(*
Nazwa:			FB_ReadWriteCSV
Opis:			Zapis uzytkownikow do pliku CSV
Wersja:			v0.1
Data:			2018-10-31
Autor:			
Urzadzenia:		
Konfiguracja:	
Info:
*)
FUNCTION_BLOCK FB_ReadWriteLogCSV
VAR
	sCSVLine				: T_MaxString := '';(* Single CSV text line (row, record), we are using string as record buffer (your are able to see read fields)  *)
	sCSVField				: T_MaxString := '';(* Single CSV field value (column, record field) *)
	nRow	 				: UDINT 	:= 0;(* Row number (record) *)
	nColumn					: UDINT 	:= 0;(* Column number (record field) *)
	hFile					: UINT		:= 0;(* File handle of the source file *)
	step					: DWORD 	:= 0;
	fbFileOpen				: FB_FileOpen;(* Opens file *)
	fbFileClose				: FB_FileClose;(* Closes file *)
	fbFileGets				: FB_FileGets;(* Reads one record (line) *)
	fbReader				: FB_CSVMemBufferReader;(* Helper function block used to parse CSV data bytes (single record line) *)
	fbFilePuts				: FB_FilePuts;(* Writes one record (line) *)
	fbWriter				: FB_CSVMemBufferWriter;(* Helper function block used to create CSV data bytes (single record line) *)
	database				: ARRAY[0..239, 0..10] OF STRING(100);(* Target PLC database *)
	i						: INT;
	iNum					: INT;
	BusyFTRIG				: F_TRIG;	// Zakonczenie zapisu/odczytu pliku
	CommandRTRIG			: R_TRIG;	// Wykrycie zapisu/odczytu
	ErrorFileDataUsers		: R_TRIG;	// Błąd zapisu/odczytu
	bNewFile				: BOOL;		// Utworzenie nowego pliku
	iMode					: INT;		// Zapis/odczyt
	
	MAX_CSV_ROWS 			: UDINT := 239;
	MAX_CSV_COLUMNS 		: UDINT := 10;
	MAX_CSV_FIELD_LENGTH	: UDINT := 100;
	
//	fbGetDateTime			: NT_GetTime;
	sDateTime				: STRING[200];
	fbFileTell				: FB_FileTell;
	fbEOF					: FB_EOF;
	fbFileSeek				: FB_FileSeek;
	
	sLineToWrite			:STRING(255);
END_VAR
	
VAR_INPUT
	bRead					: BOOL;		//Sygnal odczytu pliku
	bWrite					: BOOL;		//Sygnal zapisu pliku
	stDataArray				: ARRAY [0..239] OF S_LogData;	//Tablica z danymi
	sNetId					: T_AmsNetId := '';	(* TwinCAT system network address *)
	sFileName				: T_MaxString ;(* CSV destination file path and name *)
END_VAR
VAR_OUTPUT
	bError					: BOOL;		// Sygnal błedu
	bBusy					: BOOL;		// Sygnal zajetosci
	bDone					: BOOL;		// Sygnal zakonczenia odczytu/zapisu
	nErrId					: UDINT;	// Numer bledu
END_VAR

CASE step OF
	0:	(* Wait for rising edge at bWrite variable *)
		IF bWrite (*AND NOT fbGetDateTime.BUSY*) THEN
			bWrite 		:= FALSE;
			bBusy 		:= TRUE;
			bError		:= FALSE;
			nErrId		:= 0;
			hFile		:= 0;
			nRow	 	:= 1;			//było 0
			nColumn		:= 0;
			step 		:= 1;
			//wybiera elementy do zapisania
			FOR iNum := 0 TO TO_INT(MAX_CSV_ROWS) DO
//				sDateTime			:=SYSTEMTIME_TO_STRING(fbGetDateTime.TIMESTR);
//				sDateTime			:=DELETE(sDateTime,11,1);	//Usuwa datę
//				sDateTime			:=LEFT(sDateTime,find(sDateTime,'.')-1); //usuwa licznik ms
				    


				//	sLineToWrite := CONCAT(WSTRING_TO_STRING(P_time.s_time_mainscreen), ',');
   		 		//	sLineToWrite := CONCAT(sLineToWrite, REAL_TO_STRING(P_ADS_SCREW.lrGripperScrewer1TorqueCV));
   		 		//	sLineToWrite := CONCAT(sLineToWrite, ',');
   		 		//	sLineToWrite := CONCAT(sLineToWrite, WSTRING_TO_STRING(gvl_recipe.s_recipe_name));
   		 		//	sLineToWrite := CONCAT(sLineToWrite, '$N');	




				database[iNum,0]		:= WSTRING_TO_STRING(P_time.s_time_mainscreen);
				database[iNum,1]		:= REAL_TO_STRING(stDataArray[iNum].arData[0]);
				database[iNum,2]		:= REAL_TO_STRING(stDataArray[iNum].arData[1]);
				database[iNum,3]		:= REAL_TO_STRING(stDataArray[iNum].arData[2]);
				database[iNum,4]		:= REAL_TO_STRING(stDataArray[iNum].arData[3]);
				database[iNum,5]		:= REAL_TO_STRING(stDataArray[iNum].arData[4]);
				database[iNum,6]		:= REAL_TO_STRING(stDataArray[iNum].arData[5]);
				database[iNum,7]		:= REAL_TO_STRING(stDataArray[iNum].arData[6]);
				database[iNum,8]		:= REAL_TO_STRING(stDataArray[iNum].arData[7]);
				database[iNum,9]		:= REAL_TO_STRING(stDataArray[iNum].arData[8]);
				database[iNum,10]		:= REAL_TO_STRING(stDataArray[iNum].arData[9]);
				
//				database[iNum,0]		:= GVL.arLogDataSave1[iNum].tTime;
//				database[iNum,1]		:= REAL_TO_STRING(GVL.arLogDataSave1[iNum].arData[0]);
//				database[iNum,2]		:= REAL_TO_STRING(GVL.arLogDataSave1[iNum].arData[1]);
//				database[iNum,3]		:= REAL_TO_STRING(GVL.arLogDataSave1[iNum].arData[2]);
//				database[iNum,4]		:= REAL_TO_STRING(GVL.arLogDataSave1[iNum].arData[3]);
//				database[iNum,5]		:= REAL_TO_STRING(GVL.arLogDataSave1[iNum].arData[4]);
//				database[iNum,6]		:= REAL_TO_STRING(GVL.arLogDataSave1[iNum].arData[5]);
//				database[iNum,7]		:= REAL_TO_STRING(GVL.arLogDataSave1[iNum].arData[6]);
//				database[iNum,8]		:= REAL_TO_STRING(GVL.arLogDataSave1[iNum].arData[7]);
//				database[iNum,9]		:= REAL_TO_STRING(GVL.arLogDataSave1[iNum].arData[8]);
//				database[iNum,10]		:= REAL_TO_STRING(GVL.arLogDataSave1[iNum].arData[9]);
			END_FOR
			//zmienia . na , żeby szybciej przetwarzać dane w excelu
//			FOR i:=1 TO UDINT_TO_INT(MAX_CSV_COLUMNS) BY 1 DO
//				database[1,i]:=REPLACE(database[1,i],',',1,FIND(database[1,i],'.'));
//			END_FOR
		END_IF
	1:	(* Open source file *)
		fbFileOpen(bExecute := FALSE);
		fbFiletell(bExecute := FALSE);	//potrzebne do wykrycia nowego pliku
	//	fbEOF(bExecute:=FALSE);
		fbFileSeek(bExecute:=FALSE);	//potrzebne do wykrycia nowego pliku
		fbFileOpen( 	sNetId := sNetId, sPathName := sFileName, nMode := FOPEN_MODEAPPEND OR FOPEN_MODETEXT,(* Open file in TEXT mode! *)
						ePath := PATH_GENERIC, bExecute := TRUE );
		step := 2;
	2:(* Wait until open not busy *)
		fbFileOpen( bExecute := FALSE, bError => bError, nErrID => nErrID, hFile => hFile );
		
		IF NOT fbFileOpen.bBusy THEN
			IF NOT fbFileOpen.bError THEN
				//step := 3;
				//sprawdź czy to nowy plik czy dopisujesz
				//próbuje cofnąć pointer odczytu o -2
				fbFileSeek(sNetId := sNetId,eOrigin := SEEK_END, nSeekPos:=-2, hFile := hFile, bExecute:= TRUE, tTimeout:=T#2S);
				IF NOT fbFileSeek.bBusy THEN
					//sprawdzam gdzie jest pointer
					fbFileTell(sNetId := sNetId, hFile := hFile, bExecute:= TRUE, tTimeout:=T#2S);
					IF NOT fbFileTell.bBusy THEN
						step := 3;
						//jak pointer = 0 to znaczy że zapisano nowy plik - dodaj nagłówki do Excela
						IF fbFileTell.nSeekPos = 0 THEN
							database[1,0]		:='Czas';
							database[1,1]		:= GVL_Screw.arDataLogScrew[0];
							database[1,2]		:= GVL_Screw.arDataLogScrew[1];
							database[1,3]		:= GVL_Screw.arDataLogScrew[2];
							database[1,4]		:= GVL_Screw.arDataLogScrew[3];
							database[1,5]		:= GVL_Screw.arDataLogScrew[4];
							database[1,6]		:= GVL_Screw.arDataLogScrew[5];
							database[1,7]		:= GVL_Screw.arDataLogScrew[6];
							database[1,8]		:= GVL_Screw.arDataLogScrew[7];
							database[1,9]		:= GVL_Screw.arDataLogScrew[8];
							database[1,10]		:= GVL_Screw.arDataLogScrew[9];
						END_IF
					END_IF
				END_IF
			ELSE(* Error: file not found? *)
				step := 100;
			END_IF
		END_IF
	3:(* Convert one PLC record to CSV format *)
		sCSVLine := '';
		fbWriter.eCmd := eEnumCmd_First;(* Write first field value *)
		IF nRow <= MAX_CSV_ROWS THEN
			FOR nColumn := 0 TO MAX_CSV_COLUMNS BY 1 DO
				sCSVField := STRING_TO_CSVFIELD( database[ nRow, nColumn ], FALSE );(* TODO: Get field value from your application *)
				(* Add new field to the record buffer *)
				fbWriter( 	pBuffer := ADR( sCSVLine ), cbBuffer := SIZEOF( sCSVLine ) - 1, putValue := sCSVField, pValue := 0, cbValue := 0,
							bCRLF := ( nColumn = MAX_CSV_COLUMNS ) );(* bCRLF == TRUE => Write CRLF after the last field value *)
				IF fbWriter.bOk THEN
					fbWriter.eCmd := eEnumCmd_Next;(* Write next field value *)
				ELSE(* Error *)
					step := 100;
					RETURN;
				END_IF
			END_FOR(* FOR nColumn := 0... *)
			(* FB_FilePuts adds allready CR (carriage return) to the written line.
			We have to replace the $R$L characters with $L character to avoid double CR. *)
			IF RIGHT( sCSVLine, 2 ) = '$R$L' THEN
				sCSVLine := REPLACE( sCSVLine, '$L', 2, LEN( sCSVLine ) - 1 );
			END_IF
			nRow := nRow + 1;(* Increment number of created records (rows) *)
			step := 4;(* Write record to the file *)
		ELSE(* All rows written => Close file *)
			step := 10;
		END_IF
	4:	(* Write single text line *)
		fbFilePuts( bExecute := FALSE );
		fbFilePuts( sNetId := sNetId, hFile := hFile, sLine := sCSVLine, bExecute := TRUE );
		step := 5;
	5:(* Wait until write not busy *)
		fbFilePuts( bExecute := FALSE, bError => bError, nErrID => nErrID );
		IF NOT fbFilePuts.bBusy THEN
			IF NOT fbFilePuts.bError THEN
				step := 3;(* Write next record *)
			ELSE(* Error *)
				step := 100;
			END_IF
		END_IF
	10:	(* Close source file *)
		fbFileClose( bExecute := FALSE );
		fbFileClose( sNetId := sNetId, hFile := hFile, bExecute := TRUE );
		step := 11;
	11:(* Wait until close not busy *)
		fbFileClose( bExecute := FALSE, bError => bError, nErrID => nErrID );
		IF ( NOT fbFileClose.bBusy ) THEN
			hFile := 0;
			step := 100;
		END_IF
	100: (* Error or ready step => cleanup *)
		IF ( hFile <> 0 ) THEN
			step := 10; (* Close the source file *)
		ELSE
			bBusy := FALSE;
			step := 0;	(* Ready *)
		END_IF
END_CASE
//bWriteUsers	:=FALSE;

END_FUNCTION_BLOCK

(* stored: Version 1.1.0.1, ProductVersion 3.1.4026.13, FileIdentifier 5439378c6a91be25a604dc6da3e9682db4406e88, FileSignature 62509d563612d38e546020986ddde544ae8bef56016ffed86a15ca738652ea62f55e35a1a74a97e17c8c31741ae605d76cffd2eae707b0382a35b5fddaa21a71226077fc82e9132be4da027cf5a5f02dfa53b33b70a251b23dec41743806c0e7aa795888f37aa253af017eadc2567f769c458b1d891fe3a86d8c0e199d580d3d8d7e632226e5dd6fcc342e3c90ff7bb63a806ffc74673605ad2a34be2e7311f7ae2fea7096c8cabd7ad2bbcbc256d39483cfbe148c42a385a21fdb90da736662b2466d59908985aba90e35b482772a97a79b877bc2133896642dcbaf9328f576924cc54195550a9ab5691e52a0f3121dabc815387771ca7da33b6923c19b582a
   POU FB_ReadWriteLogCSV: Id {ce2d827d-6e07-4d50-be3b-9430b1e32c16}, SpecialFunc None *)
